FUNCTION_BLOCK ABSTRACT NodeFactory IMPLEMENTS I_NodeFactory
VAR
END_VAR

METHOD ABSTRACT Create : I_Node
END_METHOD

END_FUNCTION_BLOCK

(* stored: Version 1.1.0.1, ProductVersion 3.1.4024.12
   POU NodeFactory: Id {04da50a7-58de-036b-3757-8d6436b4271f}, SpecialFunc None
   Method Create: Id {97d4ac09-63ea-06ec-3b31-d3c7623c5067} *)
